// Mitsubishi GX Works2 project: q03   PLC: Q02/Q02H

PROGRAM MAIN
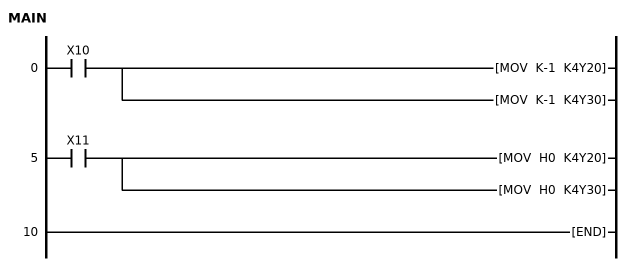
0     LD      X10
      MOV     K-1 K4Y20
      MOV     K-1 K4Y30
5     LD      X11
      MOV     H0 K4Y20
      MOV     H0 K4Y30
10    END
END_PROGRAM
